TYPE T_TransportTube : UINT; END_TYPE

(* stored: Version 1.1.0.1, ProductVersion 3.1.4022.17
   DUT T_TransportTube: Id {39aed121-ba92-4c86-a28b-34f6e10d06c2} *)
